// LS Electric XG5000 project: fda
// PLC LSPLC
// module base 0 slot 0: 입출력 모듈:XBC-DR32H (DC 24V 입력, 릴레이 출력 32점)

PROGRAM NewProgram (task: 스캔 프로그램)

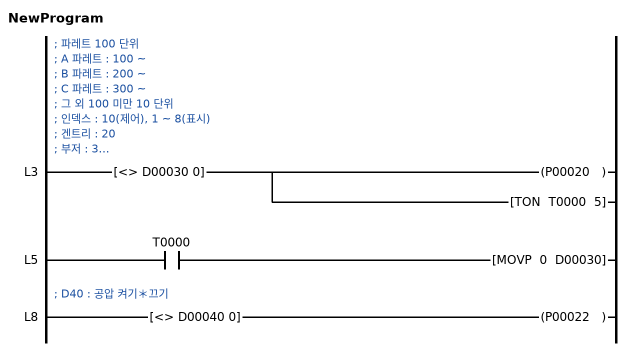
// 파레트 100 단위
// A 파레트 : 100 ~
// B 파레트 : 200 ~
// C 파레트 : 300 ~
// 
// 그 외 100 미만 10 단위
// 인덱스 : 10(제어), 1 ~ 8(표시)
// 겐트리 : 20
// 부저 : 30
// 공압 : 40
// D30 : 부저 켜기*끄기
; L3
LOAD<>    D00030 0
OUT       P00020
TON       T0000 5
; L5
LOAD      T0000
MOVP      0 D00030
// D40 : 공압 켜기＊끄기
; L8
LOAD<>    D00040 0
OUT       P00022